FUNCTION_BLOCK IndexedBuffer
VAR_IN_OUT
	bundlesQueue : ARRAY[*] OF Bundle;
	
	conveyor1 : ConveyorSC; //left/outer
	conveyor2 : ConveyorSC;
	conveyor3 : ConveyorSC;
	conveyor4 : ConveyorSC;
	conveyor5 : ConveyorSC;
	conveyor6 : ConveyorSC; //right/inner
END_VAR
VAR_OUTPUT
	requestedMode : ConveyorMode;
	trueMode : ConveyorMode;
END_VAR
VAR
	nextBuffer : POINTER TO IndexedBuffer; //no next buffer = junction*
	prevBuffer : POINTER TO IndexedBuffer;
	
	conveyors : ARRAY[1..CONSTS.numConveyorLines] OF POINTER TO ConveyorSC;
	iBundles : ARRAY[1..CONSTS.numConveyorLines] OF INT := [6(-1)];
	
	step : SectionTask;
END_VAR
VAR
	i : INT;
END_VAR

(*
this FB represents an indexed buffer for area 3
up to 6 bundles per buffer, 1 per conveyor line
	assumes 6 independent conveyer drivers
*)

fillConveyorsArray();
setConveyorMode();

(*
each section will read and copy the iterators from the previous buffer when ready
	buffers cannot write their iterators to the next buffer as the next buffer may still be active
*)

CASE step OF
	SectionTask.IDLE:
		requestedMode := ConveyorMode.IDLE;
	
		IF prevBuffer <> 0 THEN //if has previous buffer, get the iterators from there
			step := SEL(prevBuffer^.iteratorsAreValid(), 0, SectionTask.ALIGN);
			(*
			IF prevBuffer^.iteratorsAreValid() THEN
				step := SectionTask.ALIGN;
			END_IF
			*)
		ELSIF iteratorsAreValid() THEN //this is the first buffer - conveyor-bundle iterators should be assigned via receiveNewIndexes()
			step := SectionTask.DISCHARGE; //since bundles are already on the buffer, next step should be discharge
			
		END_IF
	(*
	SectionTask.ACTIVE:
		CASE masterConveyorTrueMode OF
			
		END_CASE
	*)
	SectionTask.ALIGN:
		requestedMode := ConveyorMode.FORWARD;
		
		IF NOT allConveyorsVacant() THEN //at least 1 conveyor is occupied
			iBundles := SEL(prevBuffer <> 0, iBundles, prevBuffer^.iBundles);
			step := SectionTask.DISCHARGE;
		END_IF
		
	SectionTask.ACTIVE: //
	
	SectionTask.DISCHARGE:		
		IF nextBuffer <> 0 THEN
			requestedMode := ConveyorMode.FORWARD;
			
			IF allConveyorsVacant() THEN //all conveyors vacant
				step := SectionTask.COMPLETE;
			END_IF
			
		ELSE //no next buffer - upcoming junction
			(*
			0 - set all conveyors to stop
			1 - stop conveyors at exit sensor
			2 - identify the conveyors which carry bundles that do not need transfer
				move those conveyors forward
				set their respective bundle iterators to 0 when vacant
				remaining occupied conveyors carry bundles that require transfer
			3 - transfer the remaining bundles in order of lowest index
				
			*)
			
		END_IF
		
		
	SectionTask.COMPLETE:
		requestedMode := ConveyorMode.IDLE;
		
		resetIterators();
		step := 0;
		
END_CASE

METHOD PROTECTED allConveyorsOccupied : BOOL
VAR_INPUT
END_VAR
VAR
	i : INT;
END_VAR
FOR i:=1 TO CONSTS.numConveyorLines BY 1 DO
	IF NOT conveyors[i]^.IsOccupied THEN
		RETURN;
	END_IF
END_FOR

allConveyorsOccupied := TRUE;
END_METHOD

METHOD PROTECTED allConveyorsVacant : BOOL
VAR_INPUT
END_VAR
VAR
	i : INT;
END_VAR
FOR i:=1 TO CONSTS.numConveyorLines BY 1 DO
	IF conveyors[i]^.IsOccupied THEN
		RETURN;
	END_IF
END_FOR

allConveyorsVacant := TRUE;
END_METHOD

METHOD PROTECTED computeLinks : BOOL
VAR_OUTPUT
	priorityRequest : ConveyorMode;
	trueMode : ConveyorMode;
END_VAR
VAR
	i : INT;
END_VAR
FOR i:=1 TO CONSTS.numConveyorLines BY 1 DO //calculate the highest priority request
	priorityRequest := MAX(priorityRequest, conveyors[i]^.requestedMode);
END_FOR

FOR i:=1 TO CONSTS.numConveyorLines BY 1 DO //set all conveyors to that highest priority request
	conveyors[i]^.setRequest(newRequest:= priorityRequest);
END_FOR
END_METHOD

METHOD connectTo : BOOL
VAR_INPUT
	next : POINTER TO IndexedBuffer;
END_VAR
nextBuffer := next;

IF next <> 0 THEN
	next^.prevBuffer := THIS;
END_IF
END_METHOD

METHOD conveyorsAtSensorExit : BOOL
VAR
	i : INT;
END_VAR
FOR i:=1 TO CONSTS.numConveyorLines BY 1 DO
	IF iBundles[i] <> -1 THEN
		
		RETURN;
	END_IF
END_FOR

conveyorsAtSensorExit := TRUE;
END_METHOD

METHOD PROTECTED fillConveyorsArray : BOOL
VAR_INPUT
END_VAR
{warning disable C0371}
conveyors[1] := ADR(conveyor1);
conveyors[2] := ADR(conveyor2);
conveyors[3] := ADR(conveyor3);
conveyors[4] := ADR(conveyor4);
conveyors[5] := ADR(conveyor5);
conveyors[6] := ADR(conveyor6);
END_METHOD

METHOD PROTECTED iteratorsAreValid : BOOL
VAR
	i : INT;
END_VAR
FOR i:=1 TO CONSTS.numConveyorLines BY 1 DO
	IF iBundles[i] <> -1 THEN
		iteratorsAreValid := TRUE;
		RETURN;
	END_IF
END_FOR
END_METHOD

METHOD receiveNewIterators : BOOL
VAR_INPUT
	iLine1 : INT;
	iLine2 : INT;
	iLine3 : INT;
	iLine4 : INT;
	iLine5 : INT;
	iLine6 : INT;
END_VAR
//6 ints containing the new array indexes of the new bundles in bundlesQueue, 1 for each respective conveyor line
//-1 indicates unused, non-negative are real indexes
iBundles[1] := iLine1;
iBundles[2] := iLine1;
iBundles[3] := iLine1;
iBundles[4] := iLine1;
iBundles[5] := iLine1;
iBundles[6] := iLine1;
END_METHOD

METHOD PROTECTED resetIterators : BOOL
VAR_INPUT
END_VAR
VAR
	i : INT;
END_VAR
FOR i:=1 TO CONSTS.numConveyorLines BY 1 DO
	iBundles[i] := -1;
END_FOR
END_METHOD

METHOD PROTECTED setConveyorMode : BOOL
VAR
	i : INT;
END_VAR
FOR i:=1 TO CONSTS.numConveyorLines BY 1 DO
	conveyors[i]^.setRequest(newRequest:= requestedMode);
END_FOR

FOR i:=1 TO CONSTS.numConveyorLines BY 1 DO
	trueMode := MAX(trueMode, conveyors[i]^.trueMode);
END_FOR
END_METHOD

END_FUNCTION_BLOCK

(* stored: Version 1.1.0.1, ProductVersion 3.1.4024.11
   POU IndexedBuffer: Id {05296bf2-cb04-45ac-92fd-055cc5e5d88c}, SpecialFunc None
   Folder Conveyors: Id {1fe3e051-cbac-4bf3-85b5-de2d27420a2c}
   Folder Hidden: Id {26a23429-fdbb-4c6c-9895-c0940a0ef45d}
   Method allConveyorsOccupied: Id {c24ea4eb-3729-426f-8508-b627694e0cbe}
   Method allConveyorsVacant: Id {842725e9-555f-4f73-83ee-f9427bf1651f}
   Method computeLinks: Id {a6ff1a02-d43e-4f20-a651-fb63e407c34c}
   Method connectTo: Id {216d5f49-06cb-4f39-bbc5-2791d64ebae8}
   Method conveyorsAtSensorExit: Id {4a4ef1e6-eef9-491e-af7f-fe134b7a25a8}
   Method fillConveyorsArray: Id {a951dee5-7153-4a73-bec3-29b5a1103a67}
   Method iteratorsAreValid: Id {789f4073-c4df-42ef-a20b-6e8a4d1c0196}
   Method receiveNewIterators: Id {148288dc-8073-48c3-bb0d-a90fb232de9f}
   Method resetIterators: Id {df840ce7-d550-4484-8304-6b194661333d}
   Method setConveyorMode: Id {03a04949-3224-4665-97cf-714d47794c97} *)
